TYPE ST_ClampingSafetyConfig :
STRUCT
    fMinimumAllowedPosition : LREAL;
    fModeSwitchVelocityMax : LREAL;
END_STRUCT
END_TYPE

(* stored: Version 1.1.0.1, ProductVersion 3.1.4026.20
   DUT ST_ClampingSafetyConfig: Id {c5f5f5bb-c6fd-45c9-83b1-234c8a4edfdf} *)
